GLOBALCONSTANTS DefaultPool_PWM_Numeric (* Numeric object pool constants (ID, Scale, Offset, Decimals) *)
  PACKAGE Uebungen::const::UT::PWM;
  VAR_GLOBAL CONSTANT
    InputNumber_PWM_DUTY_N : logiBUS::utils::conversion::phys::NumericObjectPool_S := (u16ObjId := 9000, r32Scale := 0.0122085215, i32Offset := 0, u8Decimals := 3);
    InputNumber_PWM_Value_N : logiBUS::utils::conversion::phys::NumericObjectPool_S := (u16ObjId := 9001, r32Scale := 1.0, i32Offset := 0, u8Decimals := 0);
    InputNumber_PWM_DUTY_OUT_N : logiBUS::utils::conversion::phys::NumericObjectPool_S := (u16ObjId := 9002, r32Scale := 0.0122085215, i32Offset := 0, u8Decimals := 3);
    InputNumber_THRESHOLD_N : logiBUS::utils::conversion::phys::NumericObjectPool_S := (u16ObjId := 9003, r32Scale := 0.0122085215, i32Offset := 0, u8Decimals := 3);
    InputNumber_HYSTERESIS_N : logiBUS::utils::conversion::phys::NumericObjectPool_S := (u16ObjId := 9004, r32Scale := 0.0122085215, i32Offset := 0, u8Decimals := 3);
    InputNumber_PWM_DUTY_NegScale_N : logiBUS::utils::conversion::phys::NumericObjectPool_S := (u16ObjId := 9005, r32Scale := -0.0122085, i32Offset := -8191, u8Decimals := 3);
    OutputNumber_100_N : logiBUS::utils::conversion::phys::NumericObjectPool_S := (u16ObjId := 12000, r32Scale := 1.0, i32Offset := 0, u8Decimals := 0);
    OutputNumber_8129_N : logiBUS::utils::conversion::phys::NumericObjectPool_S := (u16ObjId := 12001, r32Scale := 1.0, i32Offset := 0, u8Decimals := 0);
    OutputNumber_050_N : logiBUS::utils::conversion::phys::NumericObjectPool_S := (u16ObjId := 12002, r32Scale := 1.0, i32Offset := 0, u8Decimals := 0);
    OutputNumber_075_N : logiBUS::utils::conversion::phys::NumericObjectPool_S := (u16ObjId := 12003, r32Scale := 1.0, i32Offset := 0, u8Decimals := 0);
    OutputNumber_000_N : logiBUS::utils::conversion::phys::NumericObjectPool_S := (u16ObjId := 12004, r32Scale := 1.0, i32Offset := 0, u8Decimals := 0);
    OutputNumber_025_N : logiBUS::utils::conversion::phys::NumericObjectPool_S := (u16ObjId := 12005, r32Scale := 1.0, i32Offset := 0, u8Decimals := 0);
    NumberVariable_PWM_DUTY_NegScale_N : logiBUS::utils::conversion::phys::NumericObjectPool_S := (u16ObjId := 21000, r32Scale := -0.0122085, i32Offset := -8191, u8Decimals := 3);
    NumberVariable_PWM_Value_N : logiBUS::utils::conversion::phys::NumericObjectPool_S := (u16ObjId := 21001, r32Scale := 0.0122085215, i32Offset := 0, u8Decimals := 3);
  END_VAR
END_GLOBALCONSTANTS
(* other elements stored in the file *)
(* ACHTUNG: 'NumberVariable_PWM_Value' wird von mehreren Widgets mit unterschiedlicher Skalierung gebunden - 'InputNumber_PWM_DUTY' (scale=0.0122085215480405 offset=0 decimals=3) vs. 'InputNumber_PWM_Value' (scale=1.0 offset=0 decimals=0). Es gilt die Skalierung mit dem kleinsten |Scale|, alle Widgets muessen dieselbe Skalierung haben. *)
